# EPICS substitutions: CentralNodeApp/Db/userHost.substitutions
# Example substitutions file

file "db/dbExample1.db" {
    { user = "lpiccoliHost" }
}

file db/dbExample2.db {
    pattern { user, no, scan }
        { "lpiccoliHost", 1, "1 second" }
        { "lpiccoliHost", 2, "2 second" }
        { "lpiccoliHost", 3, "5 second" }
}
